// TIA Portal V20 export
FUNCTION_BLOCK "FB_OPC_AxisManagement"   // FB60, SCL
{ S7_Optimized_Access := 'TRUE' }
// stored: MemoryReserve 100, SetENOAutomatically false
   VAR
      sTeachButton : "FB_HmiKeysSignals";
      sAxisToTeachIndex { S7_SetPoint := 'True'} : DInt;
      sPositionToTeachIndex : DInt;
      sError { ExternalAccessible := 'False'; ExternalVisible := 'False'; ExternalWritable := 'False'} : Bool;
      sDone { ExternalAccessible := 'False'; ExternalVisible := 'False'; ExternalWritable := 'False'} : Bool;
      sState { ExternalAccessible := 'False'; ExternalVisible := 'False'; ExternalWritable := 'False'} : Word;
      sReadGUD_X_Load : "LBP_ReadGUD";
      sReadGUD_X_Unload { S7_SetPoint := 'True'} : "LBP_ReadGUD";
      sReadGUD_X_Blowing { S7_SetPoint := 'True'} : "LBP_ReadGUD";
      sReadGUD_Y_Load : "LBP_ReadGUD";
      sReadGUD_Y_Unload { S7_SetPoint := 'True'} : "LBP_ReadGUD";
      sReadGUD_Y_Blowing { S7_SetPoint := 'True'} : "LBP_ReadGUD";
      sReadGUD_B_Load : "LBP_ReadGUD";
      sReadGUD_B_Unload { S7_SetPoint := 'True'} : "LBP_ReadGUD";
      sReadGUD_B_Blowing { S7_SetPoint := 'True'} : "LBP_ReadGUD";
      sReadGUD_ZM_Safe { S7_SetPoint := 'True'} : "LBP_ReadGUD";
      sReadGUD_ZL_Safe { S7_SetPoint := 'True'} : "LBP_ReadGUD";
      sVarName { S7_SetPoint := 'True'} : String;
      sTON_On : TON_TIME;
      sTON_OFF { S7_SetPoint := 'True'} : TON_TIME;
      sPulseReadGUD { S7_SetPoint := 'True'} : Bool;
      sID : Int;
   END_VAR
   VAR_TEMP
      tIndex : Int;
   END_VAR
   VAR CONSTANT
      U1_AXIS_ID : DInt := 111;
      U2_AXIS_ID : DInt := 112;
      V_AXIS_ID : DInt := 120;
      W_AXIS_ID : DInt := 130;
      X_AXIS_ID : DInt := 210;
      Y_AXIS_ID : DInt := 220;
      ZL_AXIS_ID : DInt := 230;
      ZM_AXIS_ID : DInt := 240;
      B_AXIS_ID : DInt := 320;
      EXTERNAL_LOADER_ID : DInt := 211;
      SEMI_AUTO_ID : DInt := 212;
      EXT_OF_SAFETY_GATE_EXT_ID : DInt := 221;
      INT_OF_SAFETY_GATE_EXT_ID : DInt := 222;
      INSIDE_SAFETY_GATE_ID : DInt := 223;
      EXT_OF_SAFETY_GATE_INT_ID : DInt := 224;
      INT_OF_SAFETY_GATE_INT_ID : DInt := 225;
      PART_DETECTOR_ID : DInt := 230;
      BACKWALL_LOAD_ID : DInt := 241;
      BACKWALL_UNLOAD_ID : DInt := 242;
      BACKWALL_DETECTOR_ID : DInt := 250;
      LOADER_BLOW_TO_SHUTTLE_ID : DInt := 260;
      LOADER_BLOW_TO_SHUTTLE_1_ID : DInt := 261;
      LOADER_BLOW_TO_SHUTTLE_2_ID : DInt := 262;
      FROM_SHUTTLE_TO_LOADER_ID : DInt := 310;
      FROM_SHUTTLE_1_TO_LOADER : DInt := 311;
      FROM_SHUTTLE_2_TO_LOADER : DInt := 312;
      SAFE : DInt := 400;
      APPROACH_SHUTTLE_1 : DInt := 421;
      APPROACH_SHUTTLE_2 : DInt := 422;
      APPROACH_WORK_CLAMP : DInt := 430;
      FROM_LOADER_TO_WORK : DInt := 610;
      FROM_WORK_TO_LOADER : DInt := 620;
      LOADER_BLOW_TO_WORK : DInt := 730;
      STATION1 : Byte := 1;
   END_VAR
BEGIN
   REGION Description header 
       //==================================================================================
       // POSALUX Swiss SA / (C) Copyright 2025
       //----------------------------------------------------------------------------------
       // Title: FB_OPC_AxisManagement
       // Comment/Function: 
       // Author: Fabien WALDT
       // Engineering: TIA Portal v20
       //----------------------------------------------------------------------------------
       // Change log table:
       // Version  | Date     | Expert in charge | Changes applied
       // ---------|----------|------------------|-----------------------------------------
       // 00.00.01 | 20260109 | WFA              | First released version
       // =================================================================================
   END_REGION
   REGION Axis - Actual Values
       // Number of axis
       "DB_OPC_Axis".ActualValues.NumberOfAxes := 9;

       // Axis01_X
       #sID := 1;
       "DB_OPC_Axis".ActualValues.Axes[#sID].ActualPosition := "DB_AxisPosition".sAxis01_X."$AA_IM";
       "DB_OPC_Axis".ActualValues.Axes[#sID].AxisId := #X_AXIS_ID;
       "DB_OPC_Axis".ActualValues.Axes[#sID].StationNumber := #STATION1;
       // Axis02_Y
       #sID := #sID + 1;
       "DB_OPC_Axis".ActualValues.Axes[#sID].ActualPosition := "DB_AxisPosition".sAxis02_Y."$AA_IM";
       "DB_OPC_Axis".ActualValues.Axes[#sID].AxisId := #Y_AXIS_ID;
       "DB_OPC_Axis".ActualValues.Axes[#sID].StationNumber := #STATION1;
       // Axis03_ZM
       #sID := #sID + 1;
       "DB_OPC_Axis".ActualValues.Axes[#sID].ActualPosition := "DB_AxisPosition".sAxis03_ZM."$AA_IM";
       "DB_OPC_Axis".ActualValues.Axes[#sID].AxisId := #ZM_AXIS_ID;
       "DB_OPC_Axis".ActualValues.Axes[#sID].StationNumber := #STATION1;
       // Axis04_B
       #sID := #sID + 1;
       "DB_OPC_Axis".ActualValues.Axes[#sID].ActualPosition := "DB_AxisPosition".sAxis04_B."$AA_IM";
       "DB_OPC_Axis".ActualValues.Axes[#sID].AxisId := #B_AXIS_ID;
       "DB_OPC_Axis".ActualValues.Axes[#sID].StationNumber := #STATION1;
       // Axis05_U1
       #sID := #sID + 1;
       "DB_OPC_Axis".ActualValues.Axes[#sID].ActualPosition := "DB_AxisPosition".sAxis05_U1."$AA_IM";
       "DB_OPC_Axis".ActualValues.Axes[#sID].AxisId := #U1_AXIS_ID;
       "DB_OPC_Axis".ActualValues.Axes[#sID].StationNumber := #STATION1;
       // Axis06_U2
       #sID := #sID + 1;
       "DB_OPC_Axis".ActualValues.Axes[#sID].ActualPosition := "DB_AxisPosition".sAxis06_U2."$AA_IM";
       "DB_OPC_Axis".ActualValues.Axes[#sID].AxisId := #U2_AXIS_ID;
       "DB_OPC_Axis".ActualValues.Axes[#sID].StationNumber := #STATION1;
       // Axis07_V
       #sID := #sID + 1;
       "DB_OPC_Axis".ActualValues.Axes[#sID].ActualPosition := "DB_AxisPosition".sAxis07_V."$AA_IM";
       "DB_OPC_Axis".ActualValues.Axes[#sID].AxisId := #V_AXIS_ID;
       "DB_OPC_Axis".ActualValues.Axes[#sID].StationNumber := #STATION1;
       // Axis08_W
       #sID := #sID + 1;
       "DB_OPC_Axis".ActualValues.Axes[#sID].ActualPosition := "DB_AxisPosition".sAxis08_W."$AA_IM";
       "DB_OPC_Axis".ActualValues.Axes[#sID].AxisId := #W_AXIS_ID;
       "DB_OPC_Axis".ActualValues.Axes[#sID].StationNumber := #STATION1;
       // Axis09_ZL
       #sID := #sID + 1;
       "DB_OPC_Axis".ActualValues.Axes[#sID].ActualPosition := "DB_AxisPosition".sAxis09_ZL."$AA_IM";
       "DB_OPC_Axis".ActualValues.Axes[#sID].AxisId := #ZL_AXIS_ID;
       "DB_OPC_Axis".ActualValues.Axes[#sID].StationNumber := #STATION1;
   END_REGION

   REGION Taught Position PLC
       // Number of items
       "DB_OPC_Axis".TaughtPositions.NumberOfItems := 48;

       REGION Axis05_U1
           // External loader
           #sID := 1;
           "DB_OPC_Axis".TaughtPositions.Items[#sID].AxisId := #U1_AXIS_ID;
           "DB_OPC_Axis".TaughtPositions.Items[#sID].PositionId := #EXTERNAL_LOADER_ID;
           "DB_OPC_Axis".TaughtPositions.Items[#sID].StationNumber := #STATION1;
           "DB_OPC_Axis".TaughtPositions.Items[#sID].Value := "DB_AxisPosMachinePLC".Axis_U1.ExtLoadUnloadAuto;
           // Semi-auto
           #sID := #sID + 1;
           "DB_OPC_Axis".TaughtPositions.Items[#sID].AxisId := #U1_AXIS_ID;
           "DB_OPC_Axis".TaughtPositions.Items[#sID].PositionId := #SEMI_AUTO_ID;
           "DB_OPC_Axis".TaughtPositions.Items[#sID].StationNumber := #STATION1;
           "DB_OPC_Axis".TaughtPositions.Items[#sID].Value := "DB_AxisPosMachinePLC".Axis_U1.ExtLoadUnloadManu;
           // Ext of safety gate ext
           #sID := #sID + 1;
           "DB_OPC_Axis".TaughtPositions.Items[#sID].AxisId := #U1_AXIS_ID;
           "DB_OPC_Axis".TaughtPositions.Items[#sID].PositionId := #EXT_OF_SAFETY_GATE_EXT_ID;
           "DB_OPC_Axis".TaughtPositions.Items[#sID].StationNumber := #STATION1;
           "DB_OPC_Axis".TaughtPositions.Items[#sID].Value := "DB_AxisPosMachinePLC".Axis_U1.ExtGateExt;
           // Int of safety gate ext
           #sID := #sID + 1;
           "DB_OPC_Axis".TaughtPositions.Items[#sID].AxisId := #U1_AXIS_ID;
           "DB_OPC_Axis".TaughtPositions.Items[#sID].PositionId := #INT_OF_SAFETY_GATE_EXT_ID;
           "DB_OPC_Axis".TaughtPositions.Items[#sID].StationNumber := #STATION1;
           "DB_OPC_Axis".TaughtPositions.Items[#sID].Value := "DB_AxisPosMachinePLC".Axis_U1.IntGateExt;
           // Inside safety gate
           #sID := #sID + 1;
           "DB_OPC_Axis".TaughtPositions.Items[#sID].AxisId := #U1_AXIS_ID;
           "DB_OPC_Axis".TaughtPositions.Items[#sID].PositionId := #INSIDE_SAFETY_GATE_ID;
           "DB_OPC_Axis".TaughtPositions.Items[#sID].StationNumber := #STATION1;
           "DB_OPC_Axis".TaughtPositions.Items[#sID].Value := "DB_AxisPosMachinePLC".Axis_U1.Sas;
           // Ext of safety gate Int
           #sID := #sID + 1;
           "DB_OPC_Axis".TaughtPositions.Items[#sID].AxisId := #U1_AXIS_ID;
           "DB_OPC_Axis".TaughtPositions.Items[#sID].PositionId := #EXT_OF_SAFETY_GATE_INT_ID;
           "DB_OPC_Axis".TaughtPositions.Items[#sID].StationNumber := #STATION1;
           "DB_OPC_Axis".TaughtPositions.Items[#sID].Value := "DB_AxisPosMachinePLC".Axis_U1.ExtGateInt;
           // Int of safety gate Int
           #sID := #sID + 1;
           "DB_OPC_Axis".TaughtPositions.Items[#sID].AxisId := #U1_AXIS_ID;
           "DB_OPC_Axis".TaughtPositions.Items[#sID].PositionId := #INT_OF_SAFETY_GATE_INT_ID;
           "DB_OPC_Axis".TaughtPositions.Items[#sID].StationNumber := #STATION1;
           "DB_OPC_Axis".TaughtPositions.Items[#sID].Value := "DB_AxisPosMachinePLC".Axis_U1.IntGateInt;
           // Part detector
           #sID := #sID + 1;
           "DB_OPC_Axis".TaughtPositions.Items[#sID].AxisId := #U1_AXIS_ID;
           "DB_OPC_Axis".TaughtPositions.Items[#sID].PositionId := #PART_DETECTOR_ID;
           "DB_OPC_Axis".TaughtPositions.Items[#sID].StationNumber := #STATION1;
           "DB_OPC_Axis".TaughtPositions.Items[#sID].Value := "DB_AxisPosMachinePLC".Axis_U1.PartControl;
           // Backwall load
           #sID := #sID + 1;
           "DB_OPC_Axis".TaughtPositions.Items[#sID].AxisId := #U1_AXIS_ID;
           "DB_OPC_Axis".TaughtPositions.Items[#sID].PositionId := #BACKWALL_LOAD_ID;
           "DB_OPC_Axis".TaughtPositions.Items[#sID].StationNumber := #STATION1;
           "DB_OPC_Axis".TaughtPositions.Items[#sID].Value := "DB_AxisPosMachinePLC".Axis_U1.BwLoad;
           // Backwall unload
           #sID := #sID + 1;
           "DB_OPC_Axis".TaughtPositions.Items[#sID].AxisId := #U1_AXIS_ID;
           "DB_OPC_Axis".TaughtPositions.Items[#sID].PositionId := #BACKWALL_UNLOAD_ID;
           "DB_OPC_Axis".TaughtPositions.Items[#sID].StationNumber := #STATION1;
           "DB_OPC_Axis".TaughtPositions.Items[#sID].Value := "DB_AxisPosMachinePLC".Axis_U1.BwUnLoad;
           // Backwall detector
           #sID := #sID + 1;
           "DB_OPC_Axis".TaughtPositions.Items[#sID].AxisId := #U1_AXIS_ID;
           "DB_OPC_Axis".TaughtPositions.Items[#sID].PositionId := #BACKWALL_DETECTOR_ID;
           "DB_OPC_Axis".TaughtPositions.Items[#sID].StationNumber := #STATION1;
           "DB_OPC_Axis".TaughtPositions.Items[#sID].Value := "DB_AxisPosMachinePLC".Axis_U1.BwControl;
           // Loader blow to shuttle
           #sID := #sID + 1;
           "DB_OPC_Axis".TaughtPositions.Items[#sID].AxisId := #U1_AXIS_ID;
           "DB_OPC_Axis".TaughtPositions.Items[#sID].PositionId := #LOADER_BLOW_TO_SHUTTLE_ID;
           "DB_OPC_Axis".TaughtPositions.Items[#sID].StationNumber := #STATION1;
           "DB_OPC_Axis".TaughtPositions.Items[#sID].Value := "DB_AxisPosMachinePLC".Axis_U1.Blowing;
           // From shuttle to Loader
           #sID := #sID + 1;
           "DB_OPC_Axis".TaughtPositions.Items[#sID].AxisId := #U1_AXIS_ID;
           "DB_OPC_Axis".TaughtPositions.Items[#sID].PositionId := #FROM_SHUTTLE_TO_LOADER_ID;
           "DB_OPC_Axis".TaughtPositions.Items[#sID].StationNumber := #STATION1;
           "DB_OPC_Axis".TaughtPositions.Items[#sID].Value := "DB_AxisPosMachinePLC".Axis_U1.IntLoadUnload;
       END_REGION

       REGION Axis06_U2
           // External loader
           #sID := #sID + 1;
           "DB_OPC_Axis".TaughtPositions.Items[#sID].AxisId := #U2_AXIS_ID;
           "DB_OPC_Axis".TaughtPositions.Items[#sID].PositionId := #EXTERNAL_LOADER_ID;
           "DB_OPC_Axis".TaughtPositions.Items[#sID].StationNumber := #STATION1;
           "DB_OPC_Axis".TaughtPositions.Items[#sID].Value := "DB_AxisPosMachinePLC".Axis_U2.ExtLoadUnloadAuto;
           // Semi-auto
           #sID := #sID + 1;
           "DB_OPC_Axis".TaughtPositions.Items[#sID].AxisId := #U2_AXIS_ID;
           "DB_OPC_Axis".TaughtPositions.Items[#sID].PositionId := #SEMI_AUTO_ID;
           "DB_OPC_Axis".TaughtPositions.Items[#sID].StationNumber := #STATION1;
           "DB_OPC_Axis".TaughtPositions.Items[#sID].Value := "DB_AxisPosMachinePLC".Axis_U2.ExtLoadUnloadManu;
           // Ext of safety gate ext
           #sID := #sID + 1;
           "DB_OPC_Axis".TaughtPositions.Items[#sID].AxisId := #U2_AXIS_ID;
           "DB_OPC_Axis".TaughtPositions.Items[#sID].PositionId := #EXT_OF_SAFETY_GATE_EXT_ID;
           "DB_OPC_Axis".TaughtPositions.Items[#sID].StationNumber := #STATION1;
           "DB_OPC_Axis".TaughtPositions.Items[#sID].Value := "DB_AxisPosMachinePLC".Axis_U2.ExtGateExt;
           // Int of safety gate ext
           #sID := #sID + 1;
           "DB_OPC_Axis".TaughtPositions.Items[#sID].AxisId := #U2_AXIS_ID;
           "DB_OPC_Axis".TaughtPositions.Items[#sID].PositionId := #INT_OF_SAFETY_GATE_EXT_ID;
           "DB_OPC_Axis".TaughtPositions.Items[#sID].StationNumber := #STATION1;
           "DB_OPC_Axis".TaughtPositions.Items[#sID].Value := "DB_AxisPosMachinePLC".Axis_U2.IntGateExt;
           // Inside safety gate
           #sID := #sID + 1;
           "DB_OPC_Axis".TaughtPositions.Items[#sID].AxisId := #U2_AXIS_ID;
           "DB_OPC_Axis".TaughtPositions.Items[#sID].PositionId := #INSIDE_SAFETY_GATE_ID;
           "DB_OPC_Axis".TaughtPositions.Items[#sID].StationNumber := #STATION1;
           "DB_OPC_Axis".TaughtPositions.Items[#sID].Value := "DB_AxisPosMachinePLC".Axis_U2.Sas;
           // Ext of safety gate Int
           #sID := #sID + 1;
           "DB_OPC_Axis".TaughtPositions.Items[#sID].AxisId := #U2_AXIS_ID;
           "DB_OPC_Axis".TaughtPositions.Items[#sID].PositionId := #EXT_OF_SAFETY_GATE_INT_ID;
           "DB_OPC_Axis".TaughtPositions.Items[#sID].StationNumber := #STATION1;
           "DB_OPC_Axis".TaughtPositions.Items[#sID].Value := "DB_AxisPosMachinePLC".Axis_U2.ExtGateInt;
           // Int of safety gate Int
           #sID := #sID + 1;
           "DB_OPC_Axis".TaughtPositions.Items[#sID].AxisId := #U2_AXIS_ID;
           "DB_OPC_Axis".TaughtPositions.Items[#sID].PositionId := #INT_OF_SAFETY_GATE_INT_ID;
           "DB_OPC_Axis".TaughtPositions.Items[#sID].StationNumber := #STATION1;
           "DB_OPC_Axis".TaughtPositions.Items[#sID].Value := "DB_AxisPosMachinePLC".Axis_U2.IntGateInt;
           // Part detector
           #sID := #sID + 1;
           "DB_OPC_Axis".TaughtPositions.Items[#sID].AxisId := #U2_AXIS_ID;
           "DB_OPC_Axis".TaughtPositions.Items[#sID].PositionId := #PART_DETECTOR_ID;
           "DB_OPC_Axis".TaughtPositions.Items[#sID].StationNumber := #STATION1;
           "DB_OPC_Axis".TaughtPositions.Items[#sID].Value := "DB_AxisPosMachinePLC".Axis_U2.PartControl;
           // Backwall load
           #sID := #sID + 1;
           "DB_OPC_Axis".TaughtPositions.Items[#sID].AxisId := #U2_AXIS_ID;
           "DB_OPC_Axis".TaughtPositions.Items[#sID].PositionId := #BACKWALL_LOAD_ID;
           "DB_OPC_Axis".TaughtPositions.Items[#sID].StationNumber := #STATION1;
           "DB_OPC_Axis".TaughtPositions.Items[#sID].Value := "DB_AxisPosMachinePLC".Axis_U2.BwLoad;
           // Backwall unload
           #sID := #sID + 1;
           "DB_OPC_Axis".TaughtPositions.Items[#sID].AxisId := #U2_AXIS_ID;
           "DB_OPC_Axis".TaughtPositions.Items[#sID].PositionId := #BACKWALL_UNLOAD_ID;
           "DB_OPC_Axis".TaughtPositions.Items[#sID].StationNumber := #STATION1;
           "DB_OPC_Axis".TaughtPositions.Items[#sID].Value := "DB_AxisPosMachinePLC".Axis_U2.BwUnLoad;
           // Backwall detector
           #sID := #sID + 1;
           "DB_OPC_Axis".TaughtPositions.Items[#sID].AxisId := #U2_AXIS_ID;
           "DB_OPC_Axis".TaughtPositions.Items[#sID].PositionId := #BACKWALL_DETECTOR_ID;
           "DB_OPC_Axis".TaughtPositions.Items[#sID].StationNumber := #STATION1;
           "DB_OPC_Axis".TaughtPositions.Items[#sID].Value := "DB_AxisPosMachinePLC".Axis_U2.BwControl;
           // Loader blow to shuttle
           #sID := #sID + 1;
           "DB_OPC_Axis".TaughtPositions.Items[#sID].AxisId := #U2_AXIS_ID;
           "DB_OPC_Axis".TaughtPositions.Items[#sID].PositionId := #LOADER_BLOW_TO_SHUTTLE_ID;
           "DB_OPC_Axis".TaughtPositions.Items[#sID].StationNumber := #STATION1;
           "DB_OPC_Axis".TaughtPositions.Items[#sID].Value := "DB_AxisPosMachinePLC".Axis_U2.Blowing;
           // From shuttle to Loader
           #sID := #sID + 1;
           "DB_OPC_Axis".TaughtPositions.Items[#sID].AxisId := #U2_AXIS_ID;
           "DB_OPC_Axis".TaughtPositions.Items[#sID].PositionId := #FROM_SHUTTLE_TO_LOADER_ID;
           "DB_OPC_Axis".TaughtPositions.Items[#sID].StationNumber := #STATION1;
           "DB_OPC_Axis".TaughtPositions.Items[#sID].Value := "DB_AxisPosMachinePLC".Axis_U2.IntLoadUnload;
       END_REGION

       REGION Axis07_V
           // Loader blow to shuttle 1
           #sID := #sID + 1;
           "DB_OPC_Axis".TaughtPositions.Items[#sID].AxisId := #V_AXIS_ID;
           "DB_OPC_Axis".TaughtPositions.Items[#sID].PositionId := #LOADER_BLOW_TO_SHUTTLE_1_ID;
           "DB_OPC_Axis".TaughtPositions.Items[#sID].StationNumber := #STATION1;
           "DB_OPC_Axis".TaughtPositions.Items[#sID].Value := "DB_AxisPosMachinePLC".Axis_V.Shuttle_1.Blowing;
           // Loader blow to shuttle 2
           #sID := #sID + 1;
           "DB_OPC_Axis".TaughtPositions.Items[#sID].AxisId := #V_AXIS_ID;
           "DB_OPC_Axis".TaughtPositions.Items[#sID].PositionId := #LOADER_BLOW_TO_SHUTTLE_2_ID;
           "DB_OPC_Axis".TaughtPositions.Items[#sID].StationNumber := #STATION1;
           "DB_OPC_Axis".TaughtPositions.Items[#sID].Value := "DB_AxisPosMachinePLC".Axis_V.Shuttle_2.Blowing;
           // From shuttle 1 to loader
           #sID := #sID + 1;
           "DB_OPC_Axis".TaughtPositions.Items[#sID].AxisId := #V_AXIS_ID;
           "DB_OPC_Axis".TaughtPositions.Items[#sID].PositionId := #FROM_SHUTTLE_1_TO_LOADER;
           "DB_OPC_Axis".TaughtPositions.Items[#sID].StationNumber := #STATION1;
           "DB_OPC_Axis".TaughtPositions.Items[#sID].Value := "DB_AxisPosMachinePLC".Axis_V.Shuttle_1.LoadUnload;
           // From shuttle 2 to loader
           #sID := #sID + 1;
           "DB_OPC_Axis".TaughtPositions.Items[#sID].AxisId := #V_AXIS_ID;
           "DB_OPC_Axis".TaughtPositions.Items[#sID].PositionId := #FROM_SHUTTLE_2_TO_LOADER;
           "DB_OPC_Axis".TaughtPositions.Items[#sID].StationNumber := #STATION1;
           "DB_OPC_Axis".TaughtPositions.Items[#sID].Value := "DB_AxisPosMachinePLC".Axis_V.Shuttle_2.LoadUnload;
           // Safe
           #sID := #sID + 1;
           "DB_OPC_Axis".TaughtPositions.Items[#sID].AxisId := #V_AXIS_ID;
           "DB_OPC_Axis".TaughtPositions.Items[#sID].PositionId := #SAFE;
           "DB_OPC_Axis".TaughtPositions.Items[#sID].StationNumber := #STATION1;
           "DB_OPC_Axis".TaughtPositions.Items[#sID].Value := "DB_AxisPosMachinePLC".Axis_V.Safe;
       END_REGION

       REGION Axis08_W
           // Loader blow to shuttle 1
           #sID := #sID + 1;
           "DB_OPC_Axis".TaughtPositions.Items[#sID].AxisId := #W_AXIS_ID;
           "DB_OPC_Axis".TaughtPositions.Items[#sID].PositionId := #LOADER_BLOW_TO_SHUTTLE_1_ID;
           "DB_OPC_Axis".TaughtPositions.Items[#sID].StationNumber := #STATION1;
           "DB_OPC_Axis".TaughtPositions.Items[#sID].Value := "DB_AxisPosMachinePLC".Axis_W.Shuttle_1.Blowing;
           // Loader blow to shuttle 2
           #sID := #sID + 1;
           "DB_OPC_Axis".TaughtPositions.Items[#sID].AxisId := #W_AXIS_ID;
           "DB_OPC_Axis".TaughtPositions.Items[#sID].PositionId := #LOADER_BLOW_TO_SHUTTLE_2_ID;
           "DB_OPC_Axis".TaughtPositions.Items[#sID].StationNumber := #STATION1;
           "DB_OPC_Axis".TaughtPositions.Items[#sID].Value := "DB_AxisPosMachinePLC".Axis_W.Shuttle_2.Blowing;
           // From shuttle 1 to loader
           #sID := #sID + 1;
           "DB_OPC_Axis".TaughtPositions.Items[#sID].AxisId := #W_AXIS_ID;
           "DB_OPC_Axis".TaughtPositions.Items[#sID].PositionId := #FROM_SHUTTLE_1_TO_LOADER;
           "DB_OPC_Axis".TaughtPositions.Items[#sID].StationNumber := #STATION1;
           "DB_OPC_Axis".TaughtPositions.Items[#sID].Value := "DB_AxisPosMachinePLC".Axis_W.Shuttle_1.LoadUnload;
           // From shuttle 2 to loader
           #sID := #sID + 1;
           "DB_OPC_Axis".TaughtPositions.Items[#sID].AxisId := #W_AXIS_ID;
           "DB_OPC_Axis".TaughtPositions.Items[#sID].PositionId := #FROM_SHUTTLE_2_TO_LOADER;
           "DB_OPC_Axis".TaughtPositions.Items[#sID].StationNumber := #STATION1;
           "DB_OPC_Axis".TaughtPositions.Items[#sID].Value := "DB_AxisPosMachinePLC".Axis_W.Shuttle_2.LoadUnload;
           // Safe
           #sID := #sID + 1;
           "DB_OPC_Axis".TaughtPositions.Items[#sID].AxisId := #W_AXIS_ID;
           "DB_OPC_Axis".TaughtPositions.Items[#sID].PositionId := #SAFE;
           "DB_OPC_Axis".TaughtPositions.Items[#sID].StationNumber := #STATION1;
           "DB_OPC_Axis".TaughtPositions.Items[#sID].Value := "DB_AxisPosMachinePLC".Axis_W.Safe;
       END_REGION

       REGION Axis07_V (Fixture)
           // From loader to work
           #sID := #sID + 1;
           "DB_OPC_Axis".TaughtPositions.Items[#sID].AxisId := #V_AXIS_ID;
           "DB_OPC_Axis".TaughtPositions.Items[#sID].PositionId := #FROM_LOADER_TO_WORK;
           "DB_OPC_Axis".TaughtPositions.Items[#sID].StationNumber := #STATION1;
           "DB_OPC_Axis".TaughtPositions.Items[#sID].Value := "DB_AxisPosMachinePLC".Axis_V.Fixture.Load;
           // From work to loader
           #sID := #sID + 1;
           "DB_OPC_Axis".TaughtPositions.Items[#sID].AxisId := #V_AXIS_ID;
           "DB_OPC_Axis".TaughtPositions.Items[#sID].PositionId := #FROM_WORK_TO_LOADER;
           "DB_OPC_Axis".TaughtPositions.Items[#sID].StationNumber := #STATION1;
           "DB_OPC_Axis".TaughtPositions.Items[#sID].Value := "DB_AxisPosMachinePLC".Axis_V.Fixture.Unload;
           // Loader blow to work
           #sID := #sID + 1;
           "DB_OPC_Axis".TaughtPositions.Items[#sID].AxisId := #V_AXIS_ID;
           "DB_OPC_Axis".TaughtPositions.Items[#sID].PositionId := #LOADER_BLOW_TO_WORK;
           "DB_OPC_Axis".TaughtPositions.Items[#sID].StationNumber := #STATION1;
           "DB_OPC_Axis".TaughtPositions.Items[#sID].Value := "DB_AxisPosMachinePLC".Axis_V.Fixture.Blowing;
       END_REGION

       REGION Axis08_W (Fixture)
           // Approach work clamp NOT USED
           // #sID := #sID + 1;
           // "DB_OPC_Axis".TaughtPositions.Items[#sID].AxisId := #W_AXIS_ID;
           // "DB_OPC_Axis".TaughtPositions.Items[#sID].PositionId := #APPROACH_WORK_CLAMP;
           // "DB_OPC_Axis".TaughtPositions.Items[#sID].StationNumber := #STATION1;
           // "DB_OPC_Axis".TaughtPositions.Items[#sID].Value := "DB_AxisPosMachineNC".Axis_W.Approach;
           // From loader to work
           #sID := #sID + 1;
           "DB_OPC_Axis".TaughtPositions.Items[#sID].AxisId := #W_AXIS_ID;
           "DB_OPC_Axis".TaughtPositions.Items[#sID].PositionId := #FROM_LOADER_TO_WORK;
           "DB_OPC_Axis".TaughtPositions.Items[#sID].StationNumber := #STATION1;
           "DB_OPC_Axis".TaughtPositions.Items[#sID].Value := "DB_AxisPosMachinePLC".Axis_W.Fixture.Load;
           // From work to loader
           #sID := #sID + 1;
           "DB_OPC_Axis".TaughtPositions.Items[#sID].AxisId := #W_AXIS_ID;
           "DB_OPC_Axis".TaughtPositions.Items[#sID].PositionId := #FROM_WORK_TO_LOADER;
           "DB_OPC_Axis".TaughtPositions.Items[#sID].StationNumber := #STATION1;
           "DB_OPC_Axis".TaughtPositions.Items[#sID].Value := "DB_AxisPosMachinePLC".Axis_W.Fixture.Unload;
           // Loader blow to work
           #sID := #sID + 1;
           "DB_OPC_Axis".TaughtPositions.Items[#sID].AxisId := #W_AXIS_ID;
           "DB_OPC_Axis".TaughtPositions.Items[#sID].PositionId := #LOADER_BLOW_TO_WORK;
           "DB_OPC_Axis".TaughtPositions.Items[#sID].StationNumber := #STATION1;
           "DB_OPC_Axis".TaughtPositions.Items[#sID].Value := "DB_AxisPosMachinePLC".Axis_W.Fixture.Blowing;
       END_REGION
   END_REGION

   REGION Taught Position NC
       REGION Axis01_X
           // From loader to work
           #sID := #sID + 1;
           "DB_OPC_Axis".TaughtPositions.Items[#sID].AxisId := #X_AXIS_ID;
           "DB_OPC_Axis".TaughtPositions.Items[#sID].PositionId := #FROM_LOADER_TO_WORK;
           "DB_OPC_Axis".TaughtPositions.Items[#sID].StationNumber := #STATION1;
           "DB_OPC_Axis".TaughtPositions.Items[#sID].Value := "DB_AxisPosMachineNC".Axis_X.Load;
           // From work to loader
           #sID := #sID + 1;
           "DB_OPC_Axis".TaughtPositions.Items[#sID].AxisId := #X_AXIS_ID;
           "DB_OPC_Axis".TaughtPositions.Items[#sID].PositionId := #FROM_WORK_TO_LOADER;
           "DB_OPC_Axis".TaughtPositions.Items[#sID].StationNumber := #STATION1;
           "DB_OPC_Axis".TaughtPositions.Items[#sID].Value := "DB_AxisPosMachineNC".Axis_X.Unload;
           // Loader blow to work
           #sID := #sID + 1;
           "DB_OPC_Axis".TaughtPositions.Items[#sID].AxisId := #X_AXIS_ID;
           "DB_OPC_Axis".TaughtPositions.Items[#sID].PositionId := #LOADER_BLOW_TO_WORK;
           "DB_OPC_Axis".TaughtPositions.Items[#sID].StationNumber := #STATION1;
           "DB_OPC_Axis".TaughtPositions.Items[#sID].Value := "DB_AxisPosMachineNC".Axis_X.Blowing;
       END_REGION

       REGION Axis02_Y
           // From loader to work
           #sID := #sID + 1;
           "DB_OPC_Axis".TaughtPositions.Items[#sID].AxisId := #Y_AXIS_ID;
           "DB_OPC_Axis".TaughtPositions.Items[#sID].PositionId := #FROM_LOADER_TO_WORK;
           "DB_OPC_Axis".TaughtPositions.Items[#sID].StationNumber := #STATION1;
           "DB_OPC_Axis".TaughtPositions.Items[#sID].Value := "DB_AxisPosMachineNC".Axis_Y.Load;
           // From work to loader
           #sID := #sID + 1;
           "DB_OPC_Axis".TaughtPositions.Items[#sID].AxisId := #Y_AXIS_ID;
           "DB_OPC_Axis".TaughtPositions.Items[#sID].PositionId := #FROM_WORK_TO_LOADER;
           "DB_OPC_Axis".TaughtPositions.Items[#sID].StationNumber := #STATION1;
           "DB_OPC_Axis".TaughtPositions.Items[#sID].Value := "DB_AxisPosMachineNC".Axis_Y.Unload;
           // Loader blow to work
           #sID := #sID + 1;
           "DB_OPC_Axis".TaughtPositions.Items[#sID].AxisId := #Y_AXIS_ID;
           "DB_OPC_Axis".TaughtPositions.Items[#sID].PositionId := #LOADER_BLOW_TO_WORK;
           "DB_OPC_Axis".TaughtPositions.Items[#sID].StationNumber := #STATION1;
           "DB_OPC_Axis".TaughtPositions.Items[#sID].Value := "DB_AxisPosMachineNC".Axis_Y.Blowing;
       END_REGION

       // REGION Axis04_B Not Used
       //     // From loader to work
       //     #sID := #sID + 1;
       //     "DB_OPC_Axis".TaughtPositions.Items[#sID].AxisId := #B_AXIS_ID;
       //     "DB_OPC_Axis".TaughtPositions.Items[#sID].PositionId := #FROM_LOADER_TO_WORK;
       //     "DB_OPC_Axis".TaughtPositions.Items[#sID].StationNumber := #STATION1;
       //     "DB_OPC_Axis".TaughtPositions.Items[#sID].Value := "DB_AxisPosMachineNC".Axis_B.Load;
       //     // From work to loader
       //     #sID := #sID + 1;
       //     "DB_OPC_Axis".TaughtPositions.Items[#sID].AxisId := #B_AXIS_ID;
       //     "DB_OPC_Axis".TaughtPositions.Items[#sID].PositionId := #FROM_WORK_TO_LOADER;
       //     "DB_OPC_Axis".TaughtPositions.Items[#sID].StationNumber := #STATION1;
       //     "DB_OPC_Axis".TaughtPositions.Items[#sID].Value := "DB_AxisPosMachineNC".Axis_B.Unload;
       //     // Loader blow to work
       //     #sID := #sID + 1;
       //     "DB_OPC_Axis".TaughtPositions.Items[#sID].AxisId := #B_AXIS_ID;
       //     "DB_OPC_Axis".TaughtPositions.Items[#sID].PositionId := #LOADER_BLOW_TO_WORK;
       //     "DB_OPC_Axis".TaughtPositions.Items[#sID].StationNumber := #STATION1;
       //     "DB_OPC_Axis".TaughtPositions.Items[#sID].Value := "DB_AxisPosMachineNC".Axis_B.Blowing;
       // END_REGION


   END_REGION

   REGION Teach
       // Call button
       #sTeachButton(ioOPC := "DB_OPC_Axis".Teach.Buttons.Teach);
       #sTeachButton.sKeyDisable := "LBP_ModeGroup".E_JOG;
       #sTeachButton.sLedSWStatus := #sTeachButton.sKeySWToggleStatus;

       // Search axis index
       #sAxisToTeachIndex := 0;
       "DB_OPC_Axis".Teach.Current.ActualPosition := 0.0;
       FOR #tIndex := 1 TO "DB_OPC_Axis".ActualValues.NumberOfAxes DO
           IF "DB_OPC_Axis".ActualValues.Axes[#tIndex].AxisId = "DB_OPC_Axis".Teach.Parameters.AxisId THEN
               #sAxisToTeachIndex := #tIndex;
               "DB_OPC_Axis".Teach.Current.ActualPosition := "DB_OPC_Axis".ActualValues.Axes[#sAxisToTeachIndex].ActualPosition;
           END_IF;
       END_FOR;
       // Search position index
       #sPositionToTeachIndex := 0;
       "DB_OPC_Axis".Teach.Current.TaughtPosition := 0.0;
       FOR #tIndex := 1 TO "DB_OPC_Axis".TaughtPositions.NumberOfItems DO
           IF "DB_OPC_Axis".TaughtPositions.Items[#tIndex].AxisId = "DB_OPC_Axis".Teach.Parameters.AxisId
               AND "DB_OPC_Axis".TaughtPositions.Items[#tIndex].PositionId = "DB_OPC_Axis".Teach.Parameters.PositionId THEN
               #sPositionToTeachIndex := #tIndex;
               "DB_OPC_Axis".Teach.Current.TaughtPosition := "DB_OPC_Axis".TaughtPositions.Items[#sPositionToTeachIndex].Value;
           END_IF;
       END_FOR;

       // // If Teach Button, Copy Axis ActualPosition to TaughtPosition 
       // IF #TeachButton.KeySWToggleStatus THEN
       //     "DB_OPC_Axis".TaughtPositions.Items[#PositionToTeachIndex].Value := "DB_OPC_Axis".ActualValues.Axes[#AxisToTeachIndex].ActualPosition;
       //     #TeachButton.KeySWToggleStatus := FALSE;
       // END_IF;
   END_REGION

   REGION Copy Current values to Taught Values
       IF #sTeachButton.sKeySWToggleStatus THEN
           CASE "DB_OPC_Axis".Teach.Parameters.AxisId OF
           #U1_AXIS_ID:
               CASE "DB_OPC_Axis".Teach.Parameters.PositionId OF
                   #EXTERNAL_LOADER_ID:
                       "DB_AxisPosMachinePLC".Axis_U1.ExtLoadUnloadAuto := "DB_AxisPosition".sAxis05_U1."$AA_IM";
                   #SEMI_AUTO_ID:
                       "DB_AxisPosMachinePLC".Axis_U1.ExtLoadUnloadManu := "DB_AxisPosition".sAxis05_U1."$AA_IM";
                   #EXT_OF_SAFETY_GATE_EXT_ID:
                       "DB_AxisPosMachinePLC".Axis_U1.ExtGateExt := "DB_AxisPosition".sAxis05_U1."$AA_IM";
                   #INT_OF_SAFETY_GATE_EXT_ID:
                       "DB_AxisPosMachinePLC".Axis_U1.IntGateExt := "DB_AxisPosition".sAxis05_U1."$AA_IM";
                   #INSIDE_SAFETY_GATE_ID:
                       "DB_AxisPosMachinePLC".Axis_U1.Sas := "DB_AxisPosition".sAxis05_U1."$AA_IM";
                   #EXT_OF_SAFETY_GATE_INT_ID:
                       "DB_AxisPosMachinePLC".Axis_U1.ExtGateInt := "DB_AxisPosition".sAxis05_U1."$AA_IM";
                   #INT_OF_SAFETY_GATE_INT_ID:
                       "DB_AxisPosMachinePLC".Axis_U1.IntGateInt := "DB_AxisPosition".sAxis05_U1."$AA_IM";
                   #PART_DETECTOR_ID:
                       "DB_AxisPosMachinePLC".Axis_U1.PartControl := "DB_AxisPosition".sAxis05_U1."$AA_IM";
                   #BACKWALL_LOAD_ID:
                       "DB_AxisPosMachinePLC".Axis_U1.BwLoad := "DB_AxisPosition".sAxis05_U1."$AA_IM";
                   #BACKWALL_UNLOAD_ID:
                       "DB_AxisPosMachinePLC".Axis_U1.BwUnLoad := "DB_AxisPosition".sAxis05_U1."$AA_IM";
                   #BACKWALL_DETECTOR_ID:
                       "DB_AxisPosMachinePLC".Axis_U1.BwControl := "DB_AxisPosition".sAxis05_U1."$AA_IM";
                   #LOADER_BLOW_TO_SHUTTLE_ID:
                       "DB_AxisPosMachinePLC".Axis_U1.Blowing := "DB_AxisPosition".sAxis05_U1."$AA_IM";
                   #FROM_SHUTTLE_TO_LOADER_ID:
                       "DB_AxisPosMachinePLC".Axis_U1.IntLoadUnload := "DB_AxisPosition".sAxis05_U1."$AA_IM";
               END_CASE;
           #U2_AXIS_ID:
               CASE "DB_OPC_Axis".Teach.Parameters.PositionId OF
                   #EXTERNAL_LOADER_ID:
                       "DB_AxisPosMachinePLC".Axis_U1.ExtLoadUnloadAuto := "DB_AxisPosition".sAxis06_U2."$AA_IM";
                   #SEMI_AUTO_ID:
                       "DB_AxisPosMachinePLC".Axis_U1.ExtLoadUnloadManu := "DB_AxisPosition".sAxis06_U2."$AA_IM";
                   #EXT_OF_SAFETY_GATE_EXT_ID:
                       "DB_AxisPosMachinePLC".Axis_U1.ExtGateExt := "DB_AxisPosition".sAxis06_U2."$AA_IM";
                   #INT_OF_SAFETY_GATE_EXT_ID:
                       "DB_AxisPosMachinePLC".Axis_U1.IntGateExt := "DB_AxisPosition".sAxis06_U2."$AA_IM";
                   #INSIDE_SAFETY_GATE_ID:
                       "DB_AxisPosMachinePLC".Axis_U1.Sas := "DB_AxisPosition".sAxis06_U2."$AA_IM";
                   #EXT_OF_SAFETY_GATE_INT_ID:
                       "DB_AxisPosMachinePLC".Axis_U1.ExtGateInt := "DB_AxisPosition".sAxis06_U2."$AA_IM";
                   #INT_OF_SAFETY_GATE_INT_ID:
                       "DB_AxisPosMachinePLC".Axis_U1.IntGateInt := "DB_AxisPosition".sAxis06_U2."$AA_IM";
                   #PART_DETECTOR_ID:
                       "DB_AxisPosMachinePLC".Axis_U1.PartControl := "DB_AxisPosition".sAxis06_U2."$AA_IM";
                   #BACKWALL_LOAD_ID:
                       "DB_AxisPosMachinePLC".Axis_U1.BwLoad := "DB_AxisPosition".sAxis06_U2."$AA_IM";
                   #BACKWALL_UNLOAD_ID:
                       "DB_AxisPosMachinePLC".Axis_U1.BwUnLoad := "DB_AxisPosition".sAxis06_U2."$AA_IM";
                   #BACKWALL_DETECTOR_ID:
                       "DB_AxisPosMachinePLC".Axis_U1.BwControl := "DB_AxisPosition".sAxis06_U2."$AA_IM";
                   #LOADER_BLOW_TO_SHUTTLE_ID:
                       "DB_AxisPosMachinePLC".Axis_U1.Blowing := "DB_AxisPosition".sAxis06_U2."$AA_IM";
                   #FROM_SHUTTLE_TO_LOADER_ID:
                       "DB_AxisPosMachinePLC".Axis_U1.IntLoadUnload := "DB_AxisPosition".sAxis06_U2."$AA_IM";
               END_CASE;
           #V_AXIS_ID:
               CASE "DB_OPC_Axis".Teach.Parameters.PositionId OF
                   #LOADER_BLOW_TO_SHUTTLE_1_ID:
                       "DB_AxisPosMachinePLC".Axis_V.Shuttle_1.Blowing := "DB_AxisPosition".sAxis07_V."$AA_IM";
                   #LOADER_BLOW_TO_SHUTTLE_2_ID:
                       "DB_AxisPosMachinePLC".Axis_V.Shuttle_2.Blowing := "DB_AxisPosition".sAxis07_V."$AA_IM";
                   #FROM_SHUTTLE_1_TO_LOADER:
                       "DB_AxisPosMachinePLC".Axis_V.Shuttle_1.LoadUnload := "DB_AxisPosition".sAxis07_V."$AA_IM";
                   #FROM_SHUTTLE_2_TO_LOADER:
                       "DB_AxisPosMachinePLC".Axis_V.Shuttle_2.LoadUnload := "DB_AxisPosition".sAxis07_V."$AA_IM";
                   #SAFE:
                       "DB_AxisPosMachinePLC".Axis_V.Safe := "DB_AxisPosition".sAxis07_V."$AA_IM";

                   #FROM_LOADER_TO_WORK:
                       "DB_AxisPosMachinePLC".Axis_V.Fixture.Load := "DB_AxisPosition".sAxis07_V."$AA_IM";
                   #FROM_WORK_TO_LOADER:
                       "DB_AxisPosMachinePLC".Axis_V.Fixture.Unload := "DB_AxisPosition".sAxis07_V."$AA_IM";
                   #LOADER_BLOW_TO_WORK:
                       "DB_AxisPosMachinePLC".Axis_V.Fixture.Blowing := "DB_AxisPosition".sAxis07_V."$AA_IM";
               END_CASE;
           #W_AXIS_ID:
               CASE "DB_OPC_Axis".Teach.Parameters.PositionId OF
                   #LOADER_BLOW_TO_SHUTTLE_1_ID:
                       "DB_AxisPosMachinePLC".Axis_W.Shuttle_1.Blowing := "DB_AxisPosition".sAxis08_W."$AA_IM";
                   #LOADER_BLOW_TO_SHUTTLE_2_ID:
                       "DB_AxisPosMachinePLC".Axis_W.Shuttle_2.Blowing := "DB_AxisPosition".sAxis08_W."$AA_IM";
                   #FROM_SHUTTLE_1_TO_LOADER:
                       "DB_AxisPosMachinePLC".Axis_W.Shuttle_1.LoadUnload := "DB_AxisPosition".sAxis08_W."$AA_IM";
                   #FROM_SHUTTLE_2_TO_LOADER:
                       "DB_AxisPosMachinePLC".Axis_W.Shuttle_2.LoadUnload := "DB_AxisPosition".sAxis08_W."$AA_IM";
                   #SAFE:
                       "DB_AxisPosMachinePLC".Axis_W.Safe := "DB_AxisPosition".sAxis08_W."$AA_IM";

                   #FROM_LOADER_TO_WORK:
                       "DB_AxisPosMachinePLC".Axis_V.Fixture.Load := "DB_AxisPosition".sAxis08_W."$AA_IM";
                   #FROM_WORK_TO_LOADER:
                       "DB_AxisPosMachinePLC".Axis_V.Fixture.Unload := "DB_AxisPosition".sAxis08_W."$AA_IM";
                   #LOADER_BLOW_TO_WORK:
                       "DB_AxisPosMachinePLC".Axis_V.Fixture.Blowing := "DB_AxisPosition".sAxis08_W."$AA_IM";
               END_CASE;
           #X_AXIS_ID:
               CASE "DB_OPC_Axis".Teach.Parameters.PositionId OF
                   #FROM_LOADER_TO_WORK:
                       "DB_AxisPosMachineNC".Axis_X.Load := "DB_AxisPosition".sAxis01_X."$AA_IM";
                   #FROM_WORK_TO_LOADER:
                       "DB_AxisPosMachineNC".Axis_X.Unload := "DB_AxisPosition".sAxis01_X."$AA_IM";
                   #LOADER_BLOW_TO_WORK:
                       "DB_AxisPosMachineNC".Axis_X.Blowing := "DB_AxisPosition".sAxis01_X."$AA_IM";
               END_CASE;
           #Y_AXIS_ID:
               CASE "DB_OPC_Axis".Teach.Parameters.PositionId OF
                   #FROM_LOADER_TO_WORK:
                       "DB_AxisPosMachineNC".Axis_X.Load := "DB_AxisPosition".sAxis02_Y."$AA_IM";
                   #FROM_WORK_TO_LOADER:
                       "DB_AxisPosMachineNC".Axis_X.Unload := "DB_AxisPosition".sAxis02_Y."$AA_IM";
                   #LOADER_BLOW_TO_WORK:
                       "DB_AxisPosMachineNC".Axis_X.Blowing := "DB_AxisPosition".sAxis02_Y."$AA_IM";
               END_CASE;
           #B_AXIS_ID:
               CASE "DB_OPC_Axis".Teach.Parameters.PositionId OF
                   #FROM_LOADER_TO_WORK:
                       "DB_AxisPosMachineNC".Axis_X.Load := "DB_AxisPosition".sAxis04_B."$AA_IM";
                   #FROM_WORK_TO_LOADER:
                       "DB_AxisPosMachineNC".Axis_X.Unload := "DB_AxisPosition".sAxis04_B."$AA_IM";
                   #LOADER_BLOW_TO_WORK:
                       "DB_AxisPosMachineNC".Axis_X.Blowing := "DB_AxisPosition".sAxis04_B."$AA_IM";
               END_CASE;
       END_CASE;
       #sTeachButton.sKeySWToggleStatus := FALSE;
     END_IF;
   END_REGION

   REGION Read NC Position

       // TON phase ON (5 secondes)
       #sTON_On(
              IN := #sPulseReadGUD,
              PT := T#5s);

       // TON phase OFF (5 secondes)
       #sTON_OFF(
               IN := NOT #sPulseReadGUD,
               PT := T#5s);

      IF #sTON_On.Q THEN
           #sPulseReadGUD := FALSE;
       END_IF;

       IF #sTON_OFF.Q THEN
           #sPulseReadGUD := TRUE;
       END_IF;


       REGION X Axis
           #sVarName := 'CH_X_LOAD';

           #sReadGUD_X_Load(Req := #sPulseReadGUD,
                           Addr := #sVarName,
                           Area := 2,
                           Unit := 1,
                           Index1 := 0,
                           Index2 := 0,
                           CnvtToken := FALSE,
                           VarToken := NULL,
                           Error => #sReadGUD_X_Load.Error,
                           Done => #sReadGUD_X_Load.Done,
                           State => #sReadGUD_X_Load.State,
                           RD := "DB_AxisPosMachineNC".Axis_X.Load);

           #sVarName := 'CH_X_UNLOAD';

           #sReadGUD_X_Unload(Req := #sPulseReadGUD,
                           Addr := #sVarName,
                           Area := 2,
                           Unit := 1,
                           Index1 := 0,
                           Index2 := 0,
                           CnvtToken := FALSE,
                           VarToken := NULL,
                           Error => #sReadGUD_X_Unload.Error,
                           Done => #sReadGUD_X_Unload.Done,
                           State => #sReadGUD_X_Unload.State,
                           RD := "DB_AxisPosMachineNC".Axis_X.Unload);

           #sVarName := 'CH_X_BLOW';

           #sReadGUD_X_Blowing(Req := #sPulseReadGUD,
                                  Addr := #sVarName,
                                  Area := 2,
                                  Unit := 1,
                                  Index1 := 0,
                                  Index2 := 0,
                                  CnvtToken := FALSE,
                                  VarToken := NULL,
                                  Error => #sReadGUD_X_Blowing.Error,
                                  Done => #sReadGUD_X_Blowing.Done,
                                  State => #sReadGUD_X_Blowing.State,
                                  RD := "DB_AxisPosMachineNC".Axis_X.Blowing);
       END_REGION
       REGION Y Axis
           #sVarName := 'CH_Y_LOAD';

           #sReadGUD_Y_Load(Req := NOT #sPulseReadGUD,
                           Addr := #sVarName,
                           Area := 2,
                           Unit := 1,
                           Index1 := 0,
                           Index2 := 0,
                           CnvtToken := FALSE,
                           VarToken := NULL,
                           Error => #sReadGUD_Y_Load.Error,
                           Done => #sReadGUD_Y_Load.Done,
                           State => #sReadGUD_Y_Load.State,
                           RD := "DB_AxisPosMachineNC".Axis_Y.Load);

           #sVarName := 'CH_Y_UNLOAD';

           #sReadGUD_Y_Unload(Req := NOT #sPulseReadGUD,
                             Addr := #sVarName,
                             Area := 2,
                             Unit := 1,
                             Index1 := 0,
                             Index2 := 0,
                             CnvtToken := FALSE,
                             VarToken := NULL,
                             Error => #sReadGUD_Y_Unload.Error,
                             Done => #sReadGUD_Y_Unload.Done,
                             State => #sReadGUD_Y_Unload.State,
                             RD := "DB_AxisPosMachineNC".Axis_Y.Unload);

           #sVarName := 'CH_Y_BLOW';

           #sReadGUD_Y_Blowing(Req := NOT #sPulseReadGUD,
                              Addr := #sVarName,
                              Area := 2,
                              Unit := 1,
                              Index1 := 0,
                              Index2 := 0,
                              CnvtToken := FALSE,
                              VarToken := NULL,
                              Error => #sReadGUD_Y_Blowing.Error,
                              Done => #sReadGUD_Y_Blowing.Done,
                              State => #sReadGUD_Y_Blowing.State,
                              RD := "DB_AxisPosMachineNC".Axis_Y.Blowing);
       END_REGION
       REGION B Axis
           #sVarName := 'CH_B_LOAD';

           #sReadGUD_B_Load(Req := #sPulseReadGUD,
                           Addr := #sVarName,
                           Area := 2,
                           Unit := 1,
                           Index1 := 0,
                           Index2 := 0,
                           CnvtToken := FALSE,
                           VarToken := NULL,
                           Error => #sReadGUD_B_Load.Error,
                           Done => #sReadGUD_B_Load.Done,
                           State => #sReadGUD_B_Load.State,
                           RD := "DB_AxisPosMachineNC".Axis_B.Load);

           #sVarName := 'CH_B_UNLOAD';

           #sReadGUD_B_Unload(Req := #sPulseReadGUD,
                             Addr := #sVarName,
                             Area := 2,
                             Unit := 1,
                             Index1 := 0,
                             Index2 := 0,
                             CnvtToken := FALSE,
                             VarToken := NULL,
                             Error => #sReadGUD_B_Unload.Error,
                             Done => #sReadGUD_B_Unload.Done,
                             State => #sReadGUD_B_Unload.State,
                             RD := "DB_AxisPosMachineNC".Axis_B.Unload);

           #sVarName := 'CH_B_BLOW';

           #sReadGUD_B_Blowing(Req := #sPulseReadGUD,
                              Addr := #sVarName,
                              Area := 2,
                              Unit := 1,
                              Index1 := 0,
                              Index2 := 0,
                              CnvtToken := FALSE,
                              VarToken := NULL,
                              Error => #sReadGUD_B_Blowing.Error,
                              Done => #sReadGUD_B_Blowing.Done,
                              State => #sReadGUD_B_Blowing.State,
                              RD := "DB_AxisPosMachineNC".Axis_B.Blowing);
       END_REGION
       REGION ZM Axis
           #sVarName := 'CH_ZM_SAFE';

           #sReadGUD_ZM_Safe(Req := #sPulseReadGUD,
                              Addr := #sVarName,
                              Area := 2,
                              Unit := 1,
                              Index1 := 0,
                              Index2 := 0,
                              CnvtToken := FALSE,
                              VarToken := NULL,
                              Error => #sReadGUD_ZM_Safe.Error,
                              Done => #sReadGUD_ZM_Safe.Done,
                              State => #sReadGUD_ZM_Safe.State,
                              RD := "DB_AxisPosMachineNC".Axis_ZM.Safe);
         END_REGION

         REGION ZL Axis
             #sVarName := 'CH_ZL_SAFE';

             #sReadGUD_ZL_Safe(Req := NOT #sPulseReadGUD,
                              Addr := #sVarName,
                              Area := 2,
                              Unit := 1,
                              Index1 := 0,
                              Index2 := 0,
                              CnvtToken := FALSE,
                              VarToken := NULL,
                              Error => #sReadGUD_ZL_Safe.Error,
                              Done => #sReadGUD_ZL_Safe.Done,
                              State => #sReadGUD_ZL_Safe.State,
                              RD := "DB_AxisPosMachineNC".Axis_ZL.Safe);
         END_REGION
   END_REGION
END_FUNCTION_BLOCK
